// TIA Portal V19 export
FUNCTION_BLOCK "PnDiag"   // FB105, LAD
TITLE = Profinet IO Device station diagnostic
AUTHOR : PM
// Diagnostic state for IM and submodules
// stored: Access Published, MemoryReserve 100, SetENOAutomatically false
   VAR_INPUT
      HW_IODevice : HW_DEVICE;
   END_VAR
   VAR_IN_OUT
      Alarm : "PnDiag_Alr";
   END_VAR
   VAR
      IM : Struct
         Diagnostic { S7_SetPoint := 'True'} : DIS;
         "Return" : Int;
         Details : UInt;
      END_STRUCT;
      MODULES : Struct
         Diagnostic { S7_SetPoint := 'True'} : DNN;
         "Return" : Int;
         Details : UInt;
      END_STRUCT;
   END_VAR
BEGIN

REGION Network 1 (SCL): Info
   //=============================================================================
   //PM FORMING
   //-----------------------------------------------------------------------------
   // Library: StandardBlocks
   // Tested with: S7-1518TF
   // Engineering: TIA Portal V18
   // Restrictions: -
   // Requirements: S7-1500
   // Functionality: Profinet IO device diagnostic
   //
   // v1.0.0  28/12/2022 
   //=============================================================================
END_REGION

REGION Network 2: IM State
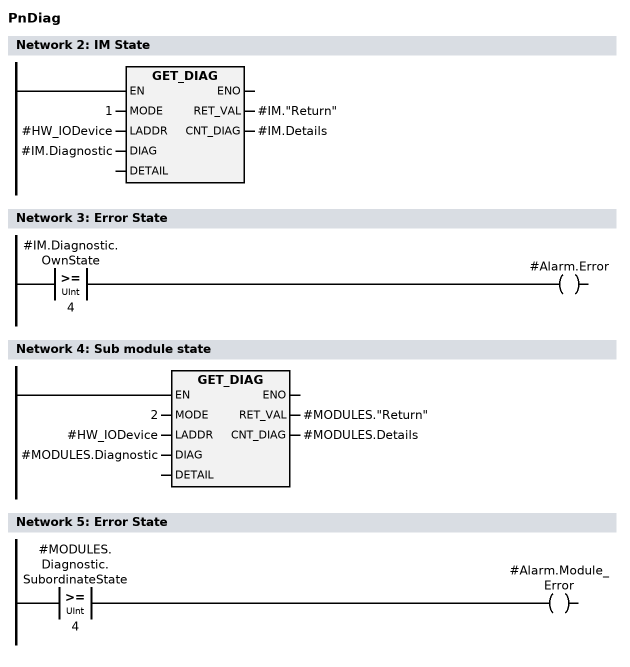
   RUNG wire#powerrail
      GET_DIAG(MODE := 1, LADDR := #HW_IODevice, DIAG := #IM.Diagnostic, DETAIL :=, RET_VAL => #IM."Return", CNT_DIAG => #IM.Details)
   END_RUNG
   // the same network as SCL:
   #IM."Return" := GET_DIAG(MODE := 1, LADDR := #HW_IODevice, DIAG := #IM.Diagnostic, CNT_DIAG => #IM.Details);
END_REGION

REGION Network 3: Error State
   RUNG wire#powerrail
      { S7_Templates := "SrcType := UInt" } GE_Contact(in1 := #IM.Diagnostic.OwnState, in2 := 4)
      Coil( #Alarm.Error )
   END_RUNG
   // the same network as SCL:
   #Alarm.Error := #IM.Diagnostic.OwnState >= 4;
END_REGION

REGION Network 4: Sub module state
   RUNG wire#powerrail
      GET_DIAG(MODE := 2, LADDR := #HW_IODevice, DIAG := #MODULES.Diagnostic, DETAIL :=, RET_VAL => #MODULES."Return", CNT_DIAG => #MODULES.Details)
   END_RUNG
   // the same network as SCL:
   #MODULES."Return" := GET_DIAG(MODE := 2,
                           LADDR := #HW_IODevice,
                           DIAG := #MODULES.Diagnostic,
                           CNT_DIAG => #MODULES.Details);
END_REGION

REGION Network 5: Error State
   RUNG wire#powerrail
      { S7_Templates := "SrcType := UInt" } GE_Contact(in1 := #MODULES.Diagnostic.SubordinateState, in2 := 4)
      Coil( #Alarm.Module_Error )
   END_RUNG
   // the same network as SCL:
   #Alarm.Module_Error := #MODULES.Diagnostic.SubordinateState >= 4;
END_REGION
END_FUNCTION_BLOCK
